PROGRAM MAIN
VAR
	readState:readState;
	State: INT;
	autoMode: autoMode;
	relaxPistons:relaxPistons;
	manualMode:manualMode;
	stateVar: INT; 
	manualModeON:BOOL;
	autoModeON: BOOL;
	allControls: BOOL;
	bmpID: STRING;
	caseImageUpdate:caseImageUpdate;
	indusoftImage: STRING;
END_VAR

readState(caseState=>State);

	autoMode(ON:=autoModeON,caseState:=State);
	
	manualMode(ON:=manualModeON, toState:=stateVar, cState:=State, prevState=>);

relaxPistons();
caseImageUpdate(id:=State,bmpID=>bmpID,indusoftImage=>indusoftImage);

END_PROGRAM

(* stored: Version 1.1.0.1, ProductVersion 3.1.4018.2
   POU MAIN: Id {1adb0c15-4940-4646-a2c2-192baed860c3}, SpecialFunc None *)
